// TIA Portal V17 export
// export: Created 2023-05-07T12:08:11.2698392Z, ExportSetting WithDefaults, DisplayName Totally Integrated Automation Portal, DisplayVersion V17, DisplayName TIA Portal Openness, DisplayVersion V17, DisplayName TIA Portal Version Control Interface, DisplayVersion V17, DisplayName TIA Portal Test Suite Advanced, DisplayVersion V17, DisplayName STEP 7 Professional, DisplayVersion V17, DisplayName SIMATIC Energy Suite, DisplayVersion V17, DisplayName STEP 7 Safety, DisplayVersion V17, DisplayName WinCC Professional, DisplayVersion V17
ORGANIZATION_BLOCK "Startup"   // OB100, LAD, Startup
TITLE = "Complete Restart"
{ S7_Optimized_Access := 'TRUE' }
VERSION : 0.1
// stored: AutoNumber true, IsIECCheckEnabled false, SetENOAutomatically false
   VAR_INPUT
      LostRetentive : Bool;   // True if retentive data are lost
      LostRTC : Bool;   // True if date and time are lost
   END_VAR
BEGIN

REGION Network 1: Call: StartupValues
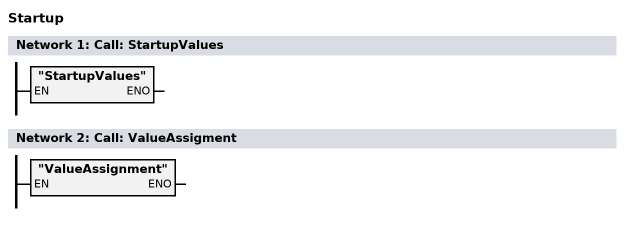
   RUNG wire#powerrail
      "StartupValues"()
   END_RUNG
   // the same network as SCL:
   "StartupValues"();
END_REGION

REGION Network 2: Call: ValueAssigment
   RUNG wire#powerrail
      "ValueAssignment"()
   END_RUNG
   // the same network as SCL:
   "ValueAssignment"();
END_REGION
END_ORGANIZATION_BLOCK
